{attribute 'qualified_only'}
VAR_GLOBAL

	Movers : ARRAY[0..38] OF AXIS_REF;
	AsseNormale: AXIS_REF;

END_VAR

(* stored: Version 1.1.0.1, ProductVersion 3.1.4024.11
   GVL GVL: Id {84cbceac-6ed6-4627-b42a-a9e2aac81071} *)
